# EPICS substitutions: iocBoot/ioc13InstekGPP_1/pid_slow.substitutions
file "$(STD)/db/pid_control.db"
{
pattern
{P,            PID,  INP,          OUT,                       LOPR,  HOPR,  DRVL,  DRVH,  PREC,   KP,  KI,   KD,  SCAN}
{13INSTEK_1:,  PID1, 13ETC_1:Ti1,  13INSTEK1:Instek1:Ch1_Vset,   0,    30,     0,    30,     3,   1.2,  1.,   0.,  ".1 second"}
{13INSTEK_1:,  PID2, 13ETC_1:Ti2,  13INSTEK1:Instek1:Ch2_Vset,   0,    30,     0,    30,     3,   1.2,  1.,   0.,  ".1 second"}
}
